# B&R Automation Studio project A2019059_Linka_Power_CP (part 31)

#### Types.typ - Local data types
```iecst
TYPE
	SkrutkovaciSetStruc : 	STRUCT
		VretenoStatus : WSTRING[80];
		VretenoFaza : USINT;
		Zasobnik : ZasobnikStruc;
		Vreteno : VretenoStruc;
		SkrutkaOdobrata : BOOL;
		SkrutkaPripravena : BOOL;
		Manual : BOOL;
		PodajSrobu : BOOL;
		CistenieVykonane : BOOL;
		VykonajCistenie : BOOL;
		Automat : BOOL;
	END_STRUCT;
	INzasobnik : 	STRUCT
		AccumulationSwitch : BOOL; (*Snimac zaplnenia S25*)
		ScrewMeasurement : BOOL; (*Kontrola matice S21*)
		FeederLevelControl : BOOL; (*Hladina v zasobniku S20*)
	END_STRUCT;
	OUTzasobnik : 	STRUCT
		StartA20 : BOOL; (*Zapnutie vibrovania A20*)
		Escapement : BOOL; (*Pustanie matky do hadice Y22*)
		FeedAir : BOOL; (*Strielanie do hadice Y21*)
		SortingAir : BOOL; (*Triedenie kusov Y30*)
		BlowOff : BOOL; (*Zhadzovanie kusov Y25*)
	END_STRUCT;
	INvreteno : 	STRUCT
		ReturnStroke : BOOL; (*Vreteno zasunute S01*)
		DeptControl : BOOL; (*Vreteno vysunute S02*)
		BrakeClosed : BOOL; (*Brzda zatvorena S13*)
		BrakeOpen : BOOL; (*Brzda otvorena S12*)
		ScrewMeasurementBrake : BOOL; (*Kontrola matice pred brzdou S15*)
		ScrewMeasurement : BOOL; (*Kontrola matice v hadici S06*)
	END_STRUCT;
	OUTvreteno : 	STRUCT
		WasteExtraction : BOOL; (*Odstranovanie spiny Y13*)
		Spindle : BOOL; (*Vysunutie vretena Y02*)
		BlastAirBrake : BOOL; (*Strielanie za brzdou Y14*)
		BrakeSpindle : BOOL; (*Brzda vretena Y12*)
		Vacuum : BOOL; (*Pridrzanie skrutky Y15*)
		CounterBlast : BOOL; (*Uvolnenie skrutky Y16*)
	END_STRUCT;
	VretenoStruc : 	STRUCT
		OUT : OUTvreteno;
		IN : INvreteno;
	END_STRUCT;
	ZasobnikStruc : 	STRUCT
		OUT : OUTzasobnik;
		IN : INzasobnik;
	END_STRUCT;
END_TYPE
```

#### Variables.var - Local variables
```iecst
VAR
	Stav_PodavacVycisteny : BOOL;
	Stav_SkrutkaM5_Pripravena : BOOL;
	SkrutkovaciSet : SkrutkovaciSetStruc;
	TprazdnyZasobnik : TON;
	TakumulaciaPlna : TON;
	TvytvorenieVakua : TON;
	TodvetranieVakua : TON;
	TprefukPredBrzdou : TON;
	TvysuvanieSpindle : TON;
	TprefukZaBrzdou : TON;
	PocetPokusovOpripravuSkrutky : USINT;
	ToddelovacZakladnaPoloha : TON;
	TpripravaSkrutky : TON;
	TodsatieNecistot : TON;
	Tvibrovanie : TON;
	TvyfukovaniePredVibrovanim : TON;
	ZapniHrniec : BOOL;
	TpodaniaSkrutky : TON;
	TpredSkrutkaPripravena : TON;
	TvypnutieOfuku : TON;
	StavSkrutkovackaVysunuta : BOOL;
	TalarmuVysunutiaSkrutkovacky : TON;
END_VAR
```

### Program Logical/Program/Pracovisko_2/P2_SkrutkovaciSet_M6 (IEC)

#### Main.st - Init, cyclic, exit code
```iecst
PROGRAM _INIT
    TprazdnyZasobnik.PT:=T#2000ms;
    TakumulaciaPlna.PT:=T#1000ms;
    TvytvorenieVakua.PT:=T#200ms;
    TodvetranieVakua.PT:=T#1s;
    TprefukPredBrzdou.PT:=T#2000ms;
    TprefukZaBrzdou.PT:=T#2000ms;
    TvysuvanieSpindle.PT:=T#1s;
    TpripravaSkrutky.PT:=T#3000ms;
    ToddelovacZakladnaPoloha.PT:=T#1000ms;
    TodsatieNecistot.PT:=T#1000ms;
    Tvibrovanie.PT:=T#3000ms;
    Stav_PodavacVycisteny:= FALSE;
    Stav_SkrutkaM6_Pripravena:= FALSE;
    TvyfukovaniePredVibrovanim.PT:= T#1000ms;
    TpodaniaSkrutky.PT:= T#1000ms;
    TpredSkrutkaPripravena.PT:= T#500ms;
    TvypnutieOfuku.PT:= T#2000ms;
    TalarmuVysunutiaSkrutkovacky.PT:= T#10s;
END_PROGRAM

PROGRAM _CYCLIC

     (********************Mapovanie IN/OUT********************************)

    SkrutkovaciSet.Manual:= P2_Srobovanie.SkrutkovaciSet_M6.Manual;
    SkrutkovaciSet.Automat:= P2_Srobovanie.SkrutkovaciSet_M6.Automat;
    SkrutkovaciSet.SkrutkaOdobrata:=P2_Srobovanie.SkrutkovaciSet_M6.SkrutkaM6_Odobrata;
    P2_Srobovanie.SkrutkovaciSet_M6.SkrutkaM6_Pripravena:= SkrutkovaciSet.SkrutkaPripravena;
    P2_Srobovanie.SkrutkovaciSet_M6.CistenieUkoncene:= SkrutkovaciSet.CistenieVykonane;
    SkrutkovaciSet.VykonajCistenie:= P2_Srobovanie.SkrutkovaciSet_M6.Cistenie;

    SkrutkovaciSet.Vreteno.IN.BrakeClosed:=P2_Srobovanie.IN.SkrutkM6_Cist_BrzdaZatvoren_MS16;
    SkrutkovaciSet.Vreteno.IN.BrakeOpen:=P2_Srobovanie.IN.SkrutkM6_Cist_BrzdaOtvorena_MS15;
    SkrutkovaciSet.Vreteno.IN.DeptControl:=P2_Srobovanie.IN.SkrutkM6_ZASUNUTY_MS14;
    SkrutkovaciSet.Vreteno.IN.ScrewMeasurement:=P2_Srobovanie.IN.SkrutkM6_SrobaPresla_IS38;
    SkrutkovaciSet.Vreteno.IN.ScrewMeasurementBrake:=P2_Srobovanie.IN.SkrutkM6_Cist_SrobaPresla_IS39;

    IF P2_Srobovanie.SkrutkovaciSet_M6.Reset AND SkrutkovaciSet.VretenoFaza <> 102 AND SkrutkovaciSet.VretenoFaza <> 104 THEN
        SkrutkovaciSet.VretenoFaza:=0;
        P2_Srobovanie.SkrutkovaciSet_M6.Reset:= FALSE;
    END_IF

    SkrutkovaciSet.Zasobnik.IN.AccumulationSwitch:=P2_Srobovanie.IN.ZasobSrobM6_ListaPLNA_OS5;
    SkrutkovaciSet.Zasobnik.IN.FeederLevelControl:=P2_Srobovanie.IN.ZasobSrobM6_PRAZDNY_IS36;
    SkrutkovaciSet.Zasobnik.IN.ScrewMeasurement:=P2_Srobovanie.IN.NastrelSrobM6_SrobaPresla_IS37;

    P2_Srobovanie.OUT.SkrutkM6_Cist_OfukVakua_RUN_YV38:=SkrutkovaciSet.Vreteno.OUT.BlastAirBrake;
    P2_Srobovanie.OUT.SkrutkM6_Cist_OTVOR_YV37:=SkrutkovaciSet.Vreteno.OUT.BrakeSpindle;
    P2_Srobovanie.OUT.SkrutkM6_OfukVakua_RUN_YV35:=SkrutkovaciSet.Vreteno.OUT.CounterBlast;
    IF SkrutkovaciSet.VretenoFaza>1 AND SkrutkovaciSet.VretenoFaza<100 THEN
        P2_Srobovanie.OUT.SkrutkM6_VYSUN_YV34:=SkrutkovaciSet.Vreteno.OUT.Spindle;
    END_IF
    P2_Srobovanie.OUT.SkrutkM6_Cist_Vakum_RUN_YV39:=SkrutkovaciSet.Vreteno.OUT.WasteExtraction;
    IF SkrutkovaciSet.VykonajCistenie THEN
        P2_Srobovanie.OUT.SkrutkM6_PrisavSkrutky_RUN_YV36:=SkrutkovaciSet.Vreteno.OUT.Vacuum;
    END_IF
    P2_Srobovanie.OUT.ZasobSrobM6_Ofuk_RUN_YV30:=SkrutkovaciSet.Zasobnik.OUT.BlowOff;
    P2_Srobovanie.OUT.NastrelSrobM6_PosunSrobu_YV32:=SkrutkovaciSet.Zasobnik.OUT.Escapement;
    P2_Srobovanie.OUT.NastrelSrobM6_NastrelSrobu_YV33:=SkrutkovaciSet.Zasobnik.OUT.FeedAir;
    P2_Srobovanie.OUT.ZasobSrobM6_OfukTried_RUN_YV31:=SkrutkovaciSet.Zasobnik.OUT.SortingAir;
    P2_Srobovanie.OUT.ZasobSrobM6_Vibrovanie_RUN_FM2:= SkrutkovaciSet.Zasobnik.OUT.StartA20;

    (********************Časáky********************************)
    TprazdnyZasobnik();
    TakumulaciaPlna();
    TvytvorenieVakua();
    TodvetranieVakua();
    TprefukPredBrzdou();
    TprefukZaBrzdou();
    TvysuvanieSpindle();
    TpripravaSkrutky();
    ToddelovacZakladnaPoloha();
    TodsatieNecistot();
    Tvibrovanie();
    TvyfukovaniePredVibrovanim();
    TpodaniaSkrutky();
    TpredSkrutkaPripravena();
    TvypnutieOfuku();
    TalarmuVysunutiaSkrutkovacky();
    (********************Zásobnik********************************)

    //kontrola akumulacie
    IF SkrutkovaciSet.Zasobnik.IN.AccumulationSwitch=1 THEN
        TakumulaciaPlna.IN:=1;
    ELSE
        TakumulaciaPlna.IN:=0;
    END_IF

    //kontrola naplnenia zasobnika
    IF SkrutkovaciSet.Zasobnik.IN.FeederLevelControl=1 THEN
        TprazdnyZasobnik.IN:=1;
    ELSE
        TprazdnyZasobnik.IN:=0;
    END_IF

    //Ovládanie vzduchov zásobníka//
    IF ZapniHrniec THEN
        IF TakumulaciaPlna.Q=1 THEN
            SkrutkovaciSet.Zasobnik.OUT.BlowOff:=1;
        ELSE
            SkrutkovaciSet.Zasobnik.OUT.BlowOff:=0;
        END_IF
        SkrutkovaciSet.Zasobnik.OUT.SortingAir:= 1;
    ELSE
        SkrutkovaciSet.Zasobnik.OUT.BlowOff:=0;
    END_IF

    IF NOT SkrutkovaciSet.Zasobnik.OUT.StartA20 AND NOT ZapniHrniec THEN
        TvypnutieOfuku.IN:= 1;
    ELSE
        TvypnutieOfuku.IN:= 0;
    END_IF

    IF EDGEPOS(TvypnutieOfuku.Q) THEN
        SkrutkovaciSet.Zasobnik.OUT.SortingAir:= 0;
    END_IF

    //ovladanie vibracneho podavaca
    IF ZapniHrniec THEN
        TvyfukovaniePredVibrovanim.IN:= 1;
    ELSE
        TvyfukovaniePredVibrovanim.IN:= 0;
    END_IF

    IF ZapniHrniec AND TvyfukovaniePredVibrovanim.Q THEN
        SkrutkovaciSet.Zasobnik.OUT.StartA20:=1;
        Tvibrovanie.IN:=1;
    ELSE
        SkrutkovaciSet.Zasobnik.OUT.StartA20:=0;
        Tvibrovanie.IN:=0;
    END_IF

    IF Tvibrovanie.Q=1 THEN
        IF TakumulaciaPlna.Q=1 AND NOT P2_Srobovanie.RR_ZapniHrniec_M6 THEN
            ZapniHrniec:= 0;
        END_IF
    END_IF

    //Zapnutie hrnca v ručnom režime//
    IF EDGEPOS(P2_Srobovanie.RR_ZapniHrniec_M6) THEN
        ZapniHrniec:= TRUE;
    END_IF
    IF EDGENEG(P2_Srobovanie.RR_ZapniHrniec_M6) THEN
        ZapniHrniec:= FALSE;
    END_IF

    //Zrušenie signálu skrutka pripravená//
    IF SkrutkovaciSet.SkrutkaPripravena=1 THEN
        IF SkrutkovaciSet.SkrutkaOdobrata=1 THEN
            SkrutkovaciSet.SkrutkaPripravena:=0;
        END_IF
    END_IF

    (********************Vreteno********************************)
    CASE SkrutkovaciSet.VretenoFaza OF
        0: SkrutkovaciSet.VretenoStatus:="Vypnute";
            SkrutkovaciSet.Vreteno.OUT.BlastAirBrake:=0;
            SkrutkovaciSet.Vreteno.OUT.BrakeSpindle:=0;
            SkrutkovaciSet.Vreteno.OUT.CounterBlast:=0;
            SkrutkovaciSet.Vreteno.OUT.Spindle:=0;
            SkrutkovaciSet.Vreteno.OUT.Vacuum:=0;
            SkrutkovaciSet.Vreteno.OUT.WasteExtraction:=0;

            SkrutkovaciSet.Zasobnik.OUT.Escapement:=0;
            SkrutkovaciSet.Zasobnik.OUT.FeedAir:=0;

            SkrutkovaciSet.Zasobnik.OUT.StartA20:=0;

            SkrutkovaciSet.CistenieVykonane:=0;
            SkrutkovaciSet.SkrutkaPripravena:=0;

            TprazdnyZasobnik.IN:=0;
            TakumulaciaPlna.IN:=0;
            TvytvorenieVakua.IN:=0;
            TodvetranieVakua.IN:=0;
            TprefukPredBrzdou.IN:=0;
            TprefukZaBrzdou.IN:=0;
            TvysuvanieSpindle.IN:=0;
            TpripravaSkrutky.IN:=0;
            ToddelovacZakladnaPoloha.IN:=0;
            TodsatieNecistot.IN:=0;
            TpodaniaSkrutky.IN:= 0;
            TpredSkrutkaPripravena.IN:= 0;
            ZapniHrniec:= 0;
            PocetPokusovOpripravuSkrutky:=0;
            StavSkrutkovackaVysunuta:= 0;
            TalarmuVysunutiaSkrutkovacky.IN:= 0;
            SkrutkovaciSet.VretenoFaza:=1;

        1: SkrutkovaciSet.VretenoStatus:="Inicializacia: cakam na povel";
            IF SkrutkovaciSet.Automat=1 THEN
                SkrutkovaciSet.CistenieVykonane:=0;
                SkrutkovaciSet.SkrutkaPripravena:=0;
                SkrutkovaciSet.VretenoFaza:=2;
            ELSIF SkrutkovaciSet.Manual=1 THEN
                SkrutkovaciSet.VretenoFaza:=250;
            END_IF

        2: SkrutkovaciSet.VretenoStatus:="Inicializacia: cakam na povel precisti hadice";

            IF SkrutkovaciSet.VykonajCistenie=1 THEN
                SkrutkovaciSet.Vreteno.OUT.Vacuum:=1;
                SkrutkovaciSet.VretenoFaza:=3;
            END_IF

        3: SkrutkovaciSet.VretenoStatus:="Inicializacia: Cakam na snimac: vreteno vysunute";
            SkrutkovaciSet.Vreteno.OUT.Spindle:=1;
            TalarmuVysunutiaSkrutkovacky.IN:= 1;

            IF P2_Srobovanie.IN.SkrutkM6_VysunutieHrotu_IOS3 > 1 THEN
                StavSkrutkovackaVysunuta:= TRUE;
                TvysuvanieSpindle.IN:=1;
            END_IF

            IF TvysuvanieSpindle.Q=1 AND StavSkrutkovackaVysunuta THEN
                TodvetranieVakua.IN:= 1;
                SkrutkovaciSet.Vreteno.OUT.CounterBlast:=1;
                SkrutkovaciSet.Vreteno.OUT.Vacuum:=0;
            END_IF

            IF TvysuvanieSpindle.Q AND StavSkrutkovackaVysunuta AND TodvetranieVakua.Q THEN
                StavSkrutkovackaVysunuta:= FALSE;
                TalarmuVysunutiaSkrutkovacky.IN:= 0;
                TvysuvanieSpindle.IN:=0;
                TodvetranieVakua.IN:= 0;
                SkrutkovaciSet.VretenoFaza:=4;
            ELSIF TalarmuVysunutiaSkrutkovacky.Q THEN
                P2_Alarmy[270]:= TRUE;
                P2_PoruchaST3:= TRUE;
            END_IF

        4: SkrutkovaciSet.VretenoStatus:="Inicializacia: Cakam na snimac: vreteno zasunute";
            SkrutkovaciSet.Vreteno.OUT.Spindle:=0;
            IF SkrutkovaciSet.Vreteno.IN.DeptControl=1 THEN
                SkrutkovaciSet.Vreteno.OUT.CounterBlast:=0;
                SkrutkovaciSet.VretenoFaza:=5;
            END_IF

        5: SkrutkovaciSet.VretenoStatus:="Inicializacia: Cakam na prefuknutie hadice za brzdou";
            TprefukZaBrzdou.IN:=1;
            SkrutkovaciSet.Vreteno.OUT.BlastAirBrake:=1;
            IF TprefukZaBrzdou.Q=1 THEN
                TprefukZaBrzdou.IN:=0;
                SkrutkovaciSet.Vreteno.OUT.BlastAirBrake:=0;
                SkrutkovaciSet.VretenoFaza:=6;
            END_IF

        6: SkrutkovaciSet.VretenoStatus:="Inicializacia: vypinam prefuk";
            TprefukZaBrzdou.IN:=0;
            SkrutkovaciSet.Vreteno.OUT.BlastAirBrake:=0;
            SkrutkovaciSet.Vreteno.OUT.Vacuum:=1;
            SkrutkovaciSet.VretenoFaza:=7;

        7: SkrutkovaciSet.VretenoStatus:="Inicializacia: Cakam na snimac: vreteno vysunute";
            SkrutkovaciSet.Vreteno.OUT.Spindle:=1;
            TalarmuVysunutiaSkrutkovacky.IN:= 1;

            IF P2_Srobovanie.IN.SkrutkM6_VysunutieHrotu_IOS3 > 1 THEN
                StavSkrutkovackaVysunuta:= TRUE;
                TvysuvanieSpindle.IN:=1;
            END_IF

            IF TvysuvanieSpindle.Q=1 AND StavSkrutkovackaVysunuta THEN
                TodvetranieVakua.IN:= 1;
                SkrutkovaciSet.Vreteno.OUT.CounterBlast:=1;
                SkrutkovaciSet.Vreteno.OUT.Vacuum:=0;
            END_IF

            IF TvysuvanieSpindle.Q AND StavSkrutkovackaVysunuta AND TodvetranieVakua.Q THEN
                StavSkrutkovackaVysunuta:= FALSE;
                TalarmuVysunutiaSkrutkovacky.IN:= 0;
                TvysuvanieSpindle.IN:=0;
                TodvetranieVakua.IN:= 0;
                SkrutkovaciSet.VretenoFaza:=8;
            ELSIF TalarmuVysunutiaSkrutkovacky.Q THEN
                P2_Alarmy[270]:= TRUE;
                P2_PoruchaST3:= TRUE;
            END_IF

        8: SkrutkovaciSet.VretenoStatus:="Inicializacia: Cakam na snimac: vreteno zasunute";
            SkrutkovaciSet.Vreteno.OUT.Spindle:=0;
            IF SkrutkovaciSet.Vreteno.IN.DeptControl=1 THEN
                SkrutkovaciSet.Vreteno.OUT.CounterBlast:=0;
                SkrutkovaciSet.VretenoFaza:=9;
            END_IF

        9: SkrutkovaciSet.VretenoStatus:="Inicializacia: Cakam na prefuknutie hadice pred brzdou";
            TprefukPredBrzdou.IN:=1;
            SkrutkovaciSet.Zasobnik.OUT.FeedAir:=1;
            IF TprefukPredBrzdou.Q=1 THEN
                TprefukPredBrzdou.IN:=0;
                SkrutkovaciSet.Zasobnik.OUT.FeedAir:=0;
                SkrutkovaciSet.VretenoFaza:=10;
            END_IF

        10: SkrutkovaciSet.VretenoStatus:="Inicializacia: Cakam na snimac: brzda uvolnena";
            SkrutkovaciSet.Vreteno.OUT.BrakeSpindle:=1;
            IF SkrutkovaciSet.Vreteno.IN.BrakeOpen=1 THEN
                SkrutkovaciSet.Vreteno.OUT.BlastAirBrake:=1;
                SkrutkovaciSet.VretenoFaza:=11;
            END_IF

        11: SkrutkovaciSet.VretenoStatus:="Inicializacia: Cakam na prefuknutie hadice za brzdou";
            TprefukZaBrzdou.IN:=1;
            SkrutkovaciSet.Vreteno.OUT.BlastAirBrake:=1;
            IF TprefukZaBrzdou.Q=1 THEN
                TprefukZaBrzdou.IN:=0;
                SkrutkovaciSet.Vreteno.OUT.BlastAirBrake:=0;
                SkrutkovaciSet.VretenoFaza:=12;
            END_IF

        12: SkrutkovaciSet.VretenoStatus:="Inicializacia: vypinam prefuk";
            TprefukZaBrzdou.IN:=0;
            SkrutkovaciSet.Vreteno.OUT.BlastAirBrake:=0;
            SkrutkovaciSet.Vreteno.OUT.Vacuum:=1;
            SkrutkovaciSet.VretenoFaza:=13;

        13: SkrutkovaciSet.VretenoStatus:="Inicializacia: Cakam na snimac: vreteno vysunute";
            SkrutkovaciSet.Vreteno.OUT.Spindle:=1;
            TalarmuVysunutiaSkrutkovacky.IN:= 1;

            IF P2_Srobovanie.IN.SkrutkM6_VysunutieHrotu_IOS3 > 1 THEN
                StavSkrutkovackaVysunuta:= TRUE;
                TvysuvanieSpindle.IN:=1;
            END_IF

            IF TvysuvanieSpindle.Q=1 AND StavSkrutkovackaVysunuta THEN
                TodvetranieVakua.IN:= 1;
                SkrutkovaciSet.Vreteno.OUT.CounterBlast:=1;
                SkrutkovaciSet.Vreteno.OUT.Vacuum:=0;
            END_IF

            IF TvysuvanieSpindle.Q AND StavSkrutkovackaVysunuta AND TodvetranieVakua.Q THEN
                StavSkrutkovackaVysunuta:= FALSE;
                TalarmuVysunutiaSkrutkovacky.IN:= 0;
                TvysuvanieSpindle.IN:=0;
                TodvetranieVakua.IN:= 0;
                SkrutkovaciSet.VretenoFaza:=14;
            ELSIF TalarmuVysunutiaSkrutkovacky.Q THEN
                P2_Alarmy[270]:= TRUE;
                P2_PoruchaST3:= TRUE;
            END_IF

        14: SkrutkovaciSet.VretenoStatus:="Inicializacia: Cakam na snimac: vreteno zasunute";
            SkrutkovaciSet.Vreteno.OUT.Spindle:=0;
            IF SkrutkovaciSet.Vreteno.IN.DeptControl=1 THEN
                SkrutkovaciSet.Vreteno.OUT.CounterBlast:=0;
                SkrutkovaciSet.VretenoFaza:=15;
            END_IF

        15: SkrutkovaciSet.VretenoStatus:="Inicializacia: Cakam na snimac: brzda zasunuta";
            SkrutkovaciSet.Vreteno.OUT.BrakeSpindle:=0;
            IF SkrutkovaciSet.Vreteno.IN.BrakeClosed=1 THEN
                SkrutkovaciSet.CistenieVykonane:=1;
                SkrutkovaciSet.VretenoFaza:=16;
            END_IF

        16: SkrutkovaciSet.VretenoStatus:="Inicializacia: Cakam na zrusenie signalu: vykonaj cistenie";
            IF SkrutkovaciSet.VykonajCistenie=0 THEN
                SkrutkovaciSet.CistenieVykonane:=0;
                SkrutkovaciSet.SkrutkaPripravena:=0;
                SkrutkovaciSet.VretenoFaza:=100;
            END_IF

        100: SkrutkovaciSet.VretenoStatus:="Cakam kym zasobnik pripravy skrutku";
            ZapniHrniec:= 1;
            IF TakumulaciaPlna.Q=1 AND SkrutkovaciSet.Zasobnik.OUT.StartA20 THEN
                TpodaniaSkrutky.IN:= 1;
            END_IF

            IF TpodaniaSkrutky.Q THEN
                TpodaniaSkrutky.IN:= 0;
                SkrutkovaciSet.VretenoFaza:=102;
            END_IF

        102: SkrutkovaciSet.VretenoStatus:="Cakam na snimac: skrutka presla hadicou";
            SkrutkovaciSet.Zasobnik.OUT.Escapement:=1;
            TpripravaSkrutky.IN:=1;
            IF SkrutkovaciSet.Zasobnik.IN.ScrewMeasurement=1 THEN
                SkrutkovaciSet.Zasobnik.OUT.FeedAir:=1;
                TpripravaSkrutky.IN:=0;
                SkrutkovaciSet.VretenoFaza:=104;
            ELSIF TpripravaSkrutky.Q=1 THEN
                TpripravaSkrutky.IN:=0;
                SkrutkovaciSet.Zasobnik.OUT.Escapement:=0;
                SkrutkovaciSet.VretenoFaza:=100;
            END_IF

        104: SkrutkovaciSet.VretenoStatus:="Cakam na snimac: skrutka presla hadicou pred brzdou";
            IF SkrutkovaciSet.Vreteno.IN.ScrewMeasurementBrake=1 THEN
                SkrutkovaciSet.Zasobnik.OUT.Escapement:=0;
                SkrutkovaciSet.Zasobnik.OUT.FeedAir:=0;
                PocetPokusovOpripravuSkrutky:=0;
                SkrutkovaciSet.VretenoFaza:=106;
            END_IF

        106: SkrutkovaciSet.VretenoStatus:="Cakam na odsatie necistot";
            SkrutkovaciSet.Vreteno.OUT.WasteExtraction:=1;
            TodsatieNecistot.IN:=1;

            IF TodsatieNecistot.Q=1 THEN
                TodsatieNecistot.IN:=0;
                SkrutkovaciSet.Vreteno.OUT.WasteExtraction:=0;
                SkrutkovaciSet.VretenoFaza:=107;
            END_IF

        107: SkrutkovaciSet.VretenoStatus:="Cakam kym skrutkovacka odoberie skrutku";
            IF SkrutkovaciSet.SkrutkaPripravena=0 AND SkrutkovaciSet.SkrutkaOdobrata=0 THEN
                SkrutkovaciSet.VretenoFaza:=108;
            END_IF

        108: SkrutkovaciSet.VretenoStatus:="Cakam na snimac: brzda uvolnena";
            SkrutkovaciSet.Vreteno.OUT.BrakeSpindle:=1;
            IF SkrutkovaciSet.Vreteno.IN.BrakeOpen=1 THEN
                SkrutkovaciSet.Vreteno.OUT.BlastAirBrake:=1;
                SkrutkovaciSet.VretenoFaza:=110;
            END_IF

        110: SkrutkovaciSet.VretenoStatus:="Cakam na snimac: skrutka presla hadicou pred vretenom";
            IF SkrutkovaciSet.Vreteno.IN.ScrewMeasurement=1 THEN
                SkrutkovaciSet.Vreteno.OUT.BlastAirBrake:=0;
                SkrutkovaciSet.Vreteno.OUT.BrakeSpindle:=0;
                SkrutkovaciSet.VretenoFaza:=112;
            END_IF

        112: SkrutkovaciSet.VretenoStatus:="Cakam na snimac: brzda zabrzdena";
            SkrutkovaciSet.Vreteno.OUT.BrakeSpindle:=0;
            IF SkrutkovaciSet.Vreteno.IN.BrakeClosed=1 AND SkrutkovaciSet.SkrutkaOdobrata=0 THEN
                TpredSkrutkaPripravena.IN:= 1;
                IF TpredSkrutkaPripravena.Q THEN
                    TpredSkrutkaPripravena.IN:= 0;
                    SkrutkovaciSet.SkrutkaPripravena:=1;
                    SkrutkovaciSet.VretenoFaza:=100;
                END_IF
            END_IF

            //*************** opakovany pokus o oddelenie skrutky *********************************

        170: SkrutkovaciSet.VretenoStatus:="Cakam na presunutie oddelovaca do zakladnej polohy";
            SkrutkovaciSet.Zasobnik.OUT.Escapement:=0;
            ToddelovacZakladnaPoloha.IN:=1;
            IF ToddelovacZakladnaPoloha.Q=1 THEN
                ToddelovacZakladnaPoloha.IN:=0;
                PocetPokusovOpripravuSkrutky:=PocetPokusovOpripravuSkrutky+1;
                IF PocetPokusovOpripravuSkrutky>3 THEN
                    PocetPokusovOpripravuSkrutky:=0;
                    SkrutkovaciSet.VretenoFaza:=171;
                ELSE
                    SkrutkovaciSet.VretenoFaza:=100;
                END_IF
            END_IF

        171: SkrutkovaciSet.VretenoStatus:="Zaseknuta skrutka v oddelovaci!!!";
    END_CASE

END_PROGRAM

PROGRAM _EXIT
	(* Insert code here *)

END_PROGRAM
```

#### Types.typ - Local data types
```iecst
TYPE
	SkrutkovaciSetStruc : 	STRUCT
		VretenoStatus : WSTRING[80];
		VretenoFaza : USINT;
		Zasobnik : ZasobnikStruc;
		Vreteno : VretenoStruc;
		SkrutkaOdobrata : BOOL;
		SkrutkaPripravena : BOOL;
		Manual : BOOL;
		PodajSrobu : BOOL;
		CistenieVykonane : BOOL;
		VykonajCistenie : BOOL;
		Automat : BOOL;
	END_STRUCT;
	INzasobnik : 	STRUCT
		AccumulationSwitch : BOOL; (*Snimac zaplnenia S25*)
		ScrewMeasurement : BOOL; (*Kontrola matice S21*)
		FeederLevelControl : BOOL; (*Hladina v zasobniku S20*)
	END_STRUCT;
	OUTzasobnik : 	STRUCT
		StartA20 : BOOL; (*Zapnutie vibrovania A20*)
		Escapement : BOOL; (*Pustanie matky do hadice Y22*)
		FeedAir : BOOL; (*Strielanie do hadice Y21*)
		SortingAir : BOOL; (*Triedenie kusov Y30*)
		BlowOff : BOOL; (*Zhadzovanie kusov Y25*)
	END_STRUCT;
	INvreteno : 	STRUCT
		ReturnStroke : BOOL; (*Vreteno zasunute S01*)
		DeptControl : BOOL; (*Vreteno vysunute S02*)
		BrakeClosed : BOOL; (*Brzda zatvorena S13*)
		BrakeOpen : BOOL; (*Brzda otvorena S12*)
		ScrewMeasurementBrake : BOOL; (*Kontrola matice pred brzdou S15*)
		ScrewMeasurement : BOOL; (*Kontrola matice v hadici S06*)
	END_STRUCT;
	OUTvreteno : 	STRUCT
		WasteExtraction : BOOL; (*Odstranovanie spiny Y13*)
		Spindle : BOOL; (*Vysunutie vretena Y02*)
		BlastAirBrake : BOOL; (*Strielanie za brzdou Y14*)
		BrakeSpindle : BOOL; (*Brzda vretena Y12*)
		Vacuum : BOOL; (*Pridrzanie skrutky Y15*)
		CounterBlast : BOOL; (*Uvolnenie skrutky Y16*)
	END_STRUCT;
	VretenoStruc : 	STRUCT
		OUT : OUTvreteno;
		IN : INvreteno;
	END_STRUCT;
	ZasobnikStruc : 	STRUCT
		OUT : OUTzasobnik;
		IN : INzasobnik;
	END_STRUCT;
END_TYPE
```

#### Variables.var - Local variables
```iecst
VAR
	Stav_PodavacVycisteny : BOOL;
	Stav_SkrutkaM6_Pripravena : BOOL;
	SkrutkovaciSet : SkrutkovaciSetStruc;
	TprazdnyZasobnik : TON;
	TakumulaciaPlna : TON;
	TvytvorenieVakua : TON;
	TodvetranieVakua : TON;
	TprefukPredBrzdou : TON;
	TvysuvanieSpindle : TON;
	TprefukZaBrzdou : TON;
	PocetPokusovOpripravuSkrutky : USINT;
	ToddelovacZakladnaPoloha : TON;
	TpripravaSkrutky : TON;
	TodsatieNecistot : TON;
	Tvibrovanie : TON;
	TvyfukovaniePredVibrovanim : TON;
	ZapniHrniec : BOOL;
	TpodaniaSkrutky : TON;
	TpredSkrutkaPripravena : TON;
	TvypnutieOfuku : TON;
	StavSkrutkovackaVysunuta : BOOL;
	TalarmuVysunutiaSkrutkovacky : TON;
END_VAR
```

### Program Logical/Program/Pracovisko_2/P2_Robot (IEC)

#### Main.st - Init, cyclic, exit code
```iecst
PROGRAM _INIT
	Triger_0:= FALSE;

END_PROGRAM

PROGRAM _CYCLIC

	//Volanie funkcie SequenceControl//
	SequenceControl(SC:= SC_P2_Robot);

	//Volanie podprogramov//
	IOLinkKomunikacia;
	ProfinetKomunikaciaRobot;

	//Reset sekcie //
	IF NOT Safety.STAV.ZonaCS_AKTIVNA THEN
		SC_P2_Robot.Step:= 0;
	ELSIF P2_PoruchaST3 AND NOT P2_StoperSrobovania.Automat AND NOT P2_StoperZvarania.Automat THEN
		SC_P2_Robot.Step:= 0;
	ELSIF P2_PoruchaST4 AND NOT P2_StoperSrobovania.Automat AND NOT P2_StoperZvarania.Automat THEN
		SC_P2_Robot.Step:= 0;
	ELSIF P2_Robot.Reset THEN
		SC_P2_Robot.Step:= 0;
		P2_Robot.Reset:= FALSE;
	END_IF

    IF NOT Safety.STAV.P2_ZonaBunky_AKTIVNA AND NOT Triger_0 THEN
        Triger_0:= TRUE;
        SC_P2_Robot.Step:= 0;
    END_IF

    IF Safety.STAV.P2_ZonaBunky_AKTIVNA THEN
        Triger_0:= FALSE;
    END_IF

	CASE SC_P2_Robot.Step OF

		0:
			SC_P2_Robot.StepName:='0 - Nulovanie';
			P2_Robot.Automat:= FALSE;
			P2_Robot.KoniecCyklu:= FALSE;
			P2_Robot.Manual:= FALSE;
			P2_Robot.Reset:= FALSE;
			P2_Robot.STAV.PoINIT:= FALSE;
			P2_Robot.KOM_OUT.Odparkovanie:= FALSE;
			P2_Robot.KOM_OUT.PP_na_Main:= FALSE;
			P2_Robot.KOM_OUT.Reset_CS:= FALSE;
			P2_Robot.KOM_OUT.StartProgramu:= FALSE;
			P2_Robot.KOM_OUT.StartProgramuMain:= FALSE;
			P2_Robot.KOM_OUT.VypniMotory:= FALSE;
			P2_Robot.KOM_OUT.ZapniMotory:= FALSE;
			IF P2_Robot.KOM_IN.Stav_RezimAUTOMAT AND P2_Robot.KOM_IN.Stav_ProgramRUN THEN
				P2_Robot.KOM_OUT.StopProgramu:= TRUE;
			ELSE
				P2_Robot.KOM_OUT.StopProgramu:= FALSE;
			END_IF
			IF Safety.STAV.ZonaCS_AKTIVNA AND Safety.STAV.P2_ZonaBunky_AKTIVNA AND NOT P2_Pracovisko.STAV.PORUCHA AND P2_Pracovisko.IN.PrivodVzduchu_SnimacTlaku_S3 AND NOT P2_Robot.KOM_IN.Stav_ProgramRUN THEN
				P2_Robot.KOM_OUT.StopProgramu:= FALSE;
				SC_P2_Robot.ResetStep:= TRUE;
				SC_P2_Robot.Step:= 1;
			END_IF

		1:
			SC_P2_Robot.StepName:='1 - Cakam na spustenie vyroby';
			P2_Robot.KoniecCyklu:= FALSE;
            IF P2_Robot.Automat THEN
				SC_P2_Robot.Step:= 2;
			ELSIF P2_Robot.Manual THEN
				SC_P2_Robot.Step:= 700;
			END_IF

		//********************************************************Inicializácia****************************************************************************//

		2:
			SC_P2_Robot.StepName:='2 - Inicializacia - cakam na spustenie inicializacie';
			SC_P2_Robot.IdleTime.PT:= T#500ms;
			SC_P2_Robot.AlarmTime.PT:= T#5s;

			SC_P2_Robot.IdleTime.IN:= TRUE;

			IF SC_P2_Robot.IdleTime.Q THEN
				SC_P2_Robot.ResetStep:= TRUE;
				SC_P2_Robot.Step:= 3;
			END_IF

		3:
			SC_P2_Robot.StepName:='2 - Inicializacia - kontrolujem central stop robota';
			SC_P2_Robot.IdleTime.PT:= T#500ms;
			SC_P2_Robot.AlarmTime.PT:= T#5s;

			IF P2_Robot.KOM_IN.Stav_RobotCS THEN
				P2_Robot.KOM_OUT.Reset_CS:= TRUE;
			END_IF

			IF NOT P2_Robot.KOM_IN.Stav_RobotCS THEN
				P2_Robot.KOM_OUT.Reset_CS:= FALSE;
				SC_P2_Robot.ResetStep:= TRUE;
				SC_P2_Robot.Step:= 4;
			END_IF

		4:
			SC_P2_Robot.StepName:='4 - Inicializacia - zapinam motory robota';
			SC_P2_Robot.IdleTime.PT:= T#5s;
            SC_P2_Robot.AlarmTime.PT:= T#5s;
            SC_P2_Robot.IdleTime.IN:= TRUE;

			IF NOT P2_Robot.KOM_IN.Stav_MotoryON THEN
				P2_Robot.KOM_OUT.ZapniMotory:= TRUE;
			END_IF

			IF P2_Robot.KOM_IN.Stav_MotoryON OR SC_P2_Robot.IdleTime.Q THEN
				P2_Robot.KOM_OUT.ZapniMotory:= FALSE;
				SC_P2_Robot.ResetStep:= TRUE;
				SC_P2_Robot.Step:= 6;
			END_IF

		6:
			SC_P2_Robot.StepName:='6 - Inicializacia - spustam program robota od zaciatku';
			SC_P2_Robot.IdleTime.PT:= T#500ms;
			SC_P2_Robot.AlarmTime.PT:= T#5s;

			IF NOT SC_P2_Robot.Switch1 THEN
				P2_Robot.KOM_OUT.StartProgramuMain:= TRUE;
				SC_P2_Robot.Switch1:= TRUE;
			END_IF

			IF P2_Robot.KOM_IN.Stav_ProgramRUN (*AND P2_Robot.KOM_IN.Stav_VystupyZresetovane*) THEN
				P2_Robot.KOM_OUT.StartProgramuMain:= FALSE;
				P2_Robot.STAV.PoINIT:= TRUE;
				SC_P2_Robot.ResetStep:= TRUE;
				SC_P2_Robot.Step:= 100;
			END_IF

			//********************************************************Automatický režim****************************************************************************//

		100:
			SC_P2_Robot.StepName:='100 - Automaticky Rezim - cakam na ukoncenie programu robota';
			SC_P2_Robot.IdleTime.PT:= T#200ms;
			SC_P2_Robot.AlarmTime.PT:= T#5s;

			IF P2_Robot.KoniecCyklu AND NOT P2_StoperSrobovania.Automat AND NOT P2_StoperZvarania.Automat AND P2_Robot.KOM_IN.Stav_RobotOdparkovany THEN
                SC_P2_Robot.ResetStep:= TRUE;
                SC_P2_Robot.Step:= 0;
            END_IF

            //*******************************************************Manuálny režim*******************************************************************************//

        700:
			SC_P2_Robot.StepName:='700 - Manualny Rezim';
			SC_P2_Robot.IdleTime.PT:= T#8s;
			SC_P2_Robot.AlarmTime.PT:= T#5s;

	END_CASE

END_PROGRAM

PROGRAM _EXIT
	(* Insert code here *)

END_PROGRAM
```

#### Variables.var - Local variables
```iecst
VAR
	Triger_0 : BOOL;
	CasOtvoreniaGripraMV : TON;
END_VAR
```

#### IOLinkKomunikacia.st
```iecst
ACTION IOLinkKomunikacia:

	//Modul ovládania gripra//
	P2_Robot.IN.GriperMvCase_Otvoreny_IS4:=	P2_Robot.PAR.Modul_IOLink_Inputs.0;
	P2_Robot.IN.GriperMvCase_DrziPowerCP_IS5:=	P2_Robot.PAR.Modul_IOLink_Inputs.1;
	P2_Robot.IN.GriperMvCase_DrziMVcase_IS6:= P2_Robot.PAR.Modul_IOLink_Inputs.2;
	P2_Robot.PAR.Modul_IOLink_Inputs.3;
	P2_Robot.PAR.Modul_IOLink_Inputs.4;
	P2_Robot.PAR.Modul_IOLink_Inputs.5;
	P2_Robot.IN.KodGripra_Bit0:= P2_Robot.PAR.Modul_IOLink_Inputs.6;
	P2_Robot.IN.KodGripra_Bit1:= P2_Robot.PAR.Modul_IOLink_Inputs.7;

	//Kodovanie griprov//
	IF P2_Robot.IN.KodGripra_Bit0 AND P2_Robot.IN.KodGripra_Bit1 THEN
		P2_Robot.KOM_OUT.TypGripra_MV:= FALSE;
		P2_Robot.KOM_OUT.TypGripra_45F:= FALSE;
		P2_Robot.KOM_OUT.TypGripra_5H:= TRUE;
	ELSIF NOT P2_Robot.IN.KodGripra_Bit0 AND P2_Robot.IN.KodGripra_Bit1 THEN
		P2_Robot.KOM_OUT.TypGripra_MV:= FALSE;
		P2_Robot.KOM_OUT.TypGripra_5H:= FALSE;
		P2_Robot.KOM_OUT.TypGripra_45F:= TRUE;
	ELSIF P2_Robot.IN.KodGripra_Bit0 AND NOT P2_Robot.IN.KodGripra_Bit1 THEN
		P2_Robot.KOM_OUT.TypGripra_5H:= FALSE;
		P2_Robot.KOM_OUT.TypGripra_45F:= FALSE;
		P2_Robot.KOM_OUT.TypGripra_MV:= TRUE;
	ELSE
		P2_Robot.KOM_OUT.TypGripra_MV:= FALSE;
		P2_Robot.KOM_OUT.TypGripra_5H:= FALSE;
		P2_Robot.KOM_OUT.TypGripra_45F:= FALSE;
	END_IF

	//Stavy griprov//
	IF P2_Robot.KOM_OUT.TypGripra_45F THEN
		IF P2_Robot.PAR.Griper_4F_5F_5H_IOLink_Inputs <= 30 THEN
			P2_Robot.KOM_OUT.Griper4F_DrziBusbary:= FALSE;
			P2_Robot.KOM_OUT.Griper4F_Zatvoreny:= FALSE;
			P2_Robot.KOM_OUT.Griper4F_Otvoreny:= TRUE;
		ELSIF P2_Robot.PAR.Griper_4F_5F_5H_IOLink_Inputs >= 803 AND P2_Robot.PAR.Griper_4F_5F_5H_IOLink_Inputs <= 900 THEN
			P2_Robot.KOM_OUT.Griper4F_Otvoreny:= FALSE;
			P2_Robot.KOM_OUT.Griper4F_Zatvoreny:= FALSE;
			P2_Robot.KOM_OUT.Griper4F_DrziBusbary:= TRUE;
		ELSIF P2_Robot.PAR.Griper_4F_5F_5H_IOLink_Inputs >= 990 THEN
			P2_Robot.KOM_OUT.Griper4F_Otvoreny:= FALSE;
			P2_Robot.KOM_OUT.Griper4F_DrziBusbary:= FALSE;
			P2_Robot.KOM_OUT.Griper4F_Zatvoreny:= TRUE;
		ELSE
			P2_Robot.KOM_OUT.Griper4F_Otvoreny:= FALSE;
			P2_Robot.KOM_OUT.Griper4F_DrziBusbary:= FALSE;
			P2_Robot.KOM_OUT.Griper4F_Zatvoreny:= FALSE;
		END_IF
	ELSIF P2_Robot.KOM_OUT.TypGripra_MV THEN
		IF P2_Robot.IN.GriperMvCase_Otvoreny_IS4 AND NOT P2_Robot.IN.GriperMvCase_DrziPowerCP_IS5 AND NOT P2_Robot.IN.GriperMvCase_DrziMVcase_IS6 THEN
			P2_Robot.KOM_OUT.GriperMvCase_DrziMVcase:= FALSE;
			P2_Robot.KOM_OUT.GriperMvCase_DrziPowerCP:= FALSE;
			P2_Robot.KOM_OUT.GriperMvCase_Zatvoreny:= FALSE;
			P2_Robot.KOM_OUT.GriperMvCase_Otvoreny:= TRUE;
		ELSIF NOT P2_Robot.IN.GriperMvCase_Otvoreny_IS4 AND P2_Robot.IN.GriperMvCase_DrziPowerCP_IS5 AND P2_Robot.IN.GriperMvCase_DrziMVcase_IS6 THEN
			P2_Robot.KOM_OUT.GriperMvCase_Otvoreny:= FALSE;
			P2_Robot.KOM_OUT.GriperMvCase_DrziPowerCP:= FALSE;
			P2_Robot.KOM_OUT.GriperMvCase_Zatvoreny:= FALSE;
			P2_Robot.KOM_OUT.GriperMvCase_DrziMVcase:= TRUE;
		ELSIF P2_Robot.IN.GriperMvCase_Otvoreny_IS4 AND P2_Robot.IN.GriperMvCase_DrziPowerCP_IS5 AND NOT P2_Robot.IN.GriperMvCase_DrziMVcase_IS6 THEN
			P2_Robot.KOM_OUT.GriperMvCase_Otvoreny:= FALSE;
			P2_Robot.KOM_OUT.GriperMvCase_DrziMVcase:= FALSE;
			P2_Robot.KOM_OUT.GriperMvCase_Zatvoreny:= FALSE;
			P2_Robot.KOM_OUT.GriperMvCase_DrziPowerCP:= TRUE;
		ELSIF NOT P2_Robot.IN.GriperMvCase_Otvoreny_IS4 AND P2_Robot.IN.GriperMvCase_DrziPowerCP_IS5 AND NOT P2_Robot.IN.GriperMvCase_DrziMVcase_IS6 THEN
			P2_Robot.KOM_OUT.GriperMvCase_Otvoreny:= FALSE;
			P2_Robot.KOM_OUT.GriperMvCase_DrziMVcase:= FALSE;
			P2_Robot.KOM_OUT.GriperMvCase_DrziPowerCP:= FALSE;
			P2_Robot.KOM_OUT.GriperMvCase_Zatvoreny:= TRUE;
		ELSE
			P2_Robot.KOM_OUT.GriperMvCase_Otvoreny:= FALSE;
			P2_Robot.KOM_OUT.GriperMvCase_DrziMVcase:= FALSE;
			P2_Robot.KOM_OUT.GriperMvCase_DrziPowerCP:= FALSE;
			P2_Robot.KOM_OUT.GriperMvCase_Zatvoreny:= FALSE;
		END_IF
	ELSIF P2_Robot.KOM_OUT.TypGripra_5H THEN
		IF P2_Robot.PAR.Griper_4F_5F_5H_IOLink_Inputs <= 30 THEN
			P2_Robot.KOM_OUT.Griper5H_Zatvoreny:= FALSE;
			P2_Robot.KOM_OUT.Griper5H_DrziBusbary:= FALSE;
			P2_Robot.KOM_OUT.Griper5H_Otvoreny:= TRUE;
		ELSIF P2_Robot.PAR.Griper_4F_5F_5H_IOLink_Inputs >= 880 AND P2_Robot.PAR.Griper_4F_5F_5H_IOLink_Inputs <= 897 THEN
			P2_Robot.KOM_OUT.Griper5H_Zatvoreny:= FALSE;
			P2_Robot.KOM_OUT.Griper5H_Otvoreny:= FALSE;
			P2_Robot.KOM_OUT.Griper5H_DrziBusbary:= TRUE;
		ELSIF P2_Robot.PAR.Griper_4F_5F_5H_IOLink_Inputs >= 992 THEN
			P2_Robot.KOM_OUT.Griper5H_Otvoreny:= FALSE;
			P2_Robot.KOM_OUT.Griper5H_DrziBusbary:= FALSE;
			P2_Robot.KOM_OUT.Griper5H_Zatvoreny:= TRUE;
		ELSE
			P2_Robot.KOM_OUT.Griper5H_Otvoreny:= FALSE;
			P2_Robot.KOM_OUT.Griper5H_DrziBusbary:= FALSE;
			P2_Robot.KOM_OUT.Griper5H_Zatvoreny:= FALSE;
		END_IF
	ELSE
		P2_Robot.KOM_OUT.Griper4F_Otvoreny:= FALSE;
		P2_Robot.KOM_OUT.Griper4F_DrziBusbary:= FALSE;
		P2_Robot.KOM_OUT.Griper4F_Zatvoreny:= FALSE;
		P2_Robot.KOM_OUT.GriperMvCase_Otvoreny:= FALSE;
		P2_Robot.KOM_OUT.GriperMvCase_DrziMVcase:= FALSE;
		P2_Robot.KOM_OUT.GriperMvCase_DrziPowerCP:= FALSE;
		P2_Robot.KOM_OUT.GriperMvCase_Zatvoreny:= FALSE;
		P2_Robot.KOM_OUT.Griper5H_Otvoreny:= FALSE;
		P2_Robot.KOM_OUT.Griper5H_DrziBusbary:= FALSE;
		P2_Robot.KOM_OUT.Griper5H_Zatvoreny:= FALSE;
	END_IF

		END_ACTION
```

#### ProfinetKomunikaciaRobot.st
```iecst
ACTION ProfinetKomunikaciaRobot:

	//Vstupy z Robota do PLC//
	P2_Robot.KOM_IN.Stav_RezimAUTOMAT:= P2_Robot.KOM_IN.Profinet_PLC_INPUTS[0].0;
	P2_Robot.KOM_IN.Stav_ProgramRUN:= P2_Robot.KOM_IN.Profinet_PLC_INPUTS[0].1;
	P2_Robot.KOM_IN.Stav_MotoryOFF:= P2_Robot.KOM_IN.Profinet_PLC_INPUTS[0].2;
	P2_Robot.KOM_IN.Stav_MotoryON:= P2_Robot.KOM_IN.Profinet_PLC_INPUTS[0].3;
	P2_Robot.KOM_IN.Stav_RobotCS:= P2_Robot.KOM_IN.Profinet_PLC_INPUTS[0].4;
	P2_Robot.KOM_IN.Profinet_PLC_INPUTS[0].5;
	P2_Robot.KOM_IN.Profinet_PLC_INPUTS[0].6;
	P2_Robot.KOM_IN.Profinet_PLC_INPUTS[0].7;

	P2_Robot.OUT.ZatvorGriper_YV4:= P2_Robot.KOM_IN.Profinet_PLC_INPUTS[1].0;
	P2_Robot.OUT.OtvorGriper_YV3:= P2_Robot.KOM_IN.Profinet_PLC_INPUTS[1].1;
	P2_Robot.OUT.ZaistiGriper_YV1:= P2_Robot.KOM_IN.Profinet_PLC_INPUTS[1].2;
	P2_Robot.OUT.OdistiGriper_YV2:= P2_Robot.KOM_IN.Profinet_PLC_INPUTS[1].3;
	P2_Robot.OUT.ZapniVakum5H_YV8:= P2_Robot.KOM_IN.Profinet_PLC_INPUTS[1].4;
	P2_Robot.OUT.ZapniVakum4F5F_YV6:= P2_Robot.KOM_IN.Profinet_PLC_INPUTS[1].5;
	P2_Robot.KOM_IN.Stav_Busbary5H_Odobrate:= P2_Robot.KOM_IN.Profinet_PLC_INPUTS[1].6;
	P2_Robot.KOM_IN.Stav_Busbary5F_Odobrate:= P2_Robot.KOM_IN.Profinet_PLC_INPUTS[1].7;

	P2_Robot.KOM_IN.Stav_Busbary4F_Odobrate:= P2_Robot.KOM_IN.Profinet_PLC_INPUTS[2].0;
	P2_Robot.KOM_IN.Stav_Busbary5H_Polozene:= P2_Robot.KOM_IN.Profinet_PLC_INPUTS[2].1;
	P2_Robot.KOM_IN.Stav_Busbary5F_Polozene:= P2_Robot.KOM_IN.Profinet_PLC_INPUTS[2].2;
	P2_Robot.KOM_IN.Stav_Busbary4F_Polozene:= P2_Robot.KOM_IN.Profinet_PLC_INPUTS[2].3;
	P2_Robot.KOM_IN.Stav_RobotPoziciaCakania:= P2_Robot.KOM_IN.Profinet_PLC_INPUTS[2].4;
	P2_Robot.KOM_IN.Stav_Filter5H_Dotlaceny:= P2_Robot.KOM_IN.Profinet_PLC_INPUTS[2].5;
	P2_Robot.KOM_IN.Profinet_PLC_INPUTS[2].6;
	P2_Robot.KOM_IN.Stav_Cistenie_PowerCP_Odobrate:= P2_Robot.KOM_IN.Profinet_PLC_INPUTS[2].7;

	P2_Robot.KOM_IN.Profinet_PLC_INPUTS[3].0;
	P2_Robot.KOM_IN.Profinet_PLC_INPUTS[3].1;
	P2_Robot.KOM_IN.Stav_Cistenie_Otacanie_Ukoncene:= P2_Robot.KOM_IN.Profinet_PLC_INPUTS[3].2;
	P2_Robot.KOM_IN.Stav_Cistenie_PowerCP_v_Cisteni:= P2_Robot.KOM_IN.Profinet_PLC_INPUTS[3].3;
	P2_Robot.KOM_IN.Stav_Cistenie_PowerCP_Polozene:= P2_Robot.KOM_IN.Profinet_PLC_INPUTS[3].4;
	P2_Robot.KOM_IN.Profinet_PLC_INPUTS[3].5;
	P2_Robot.KOM_IN.Profinet_PLC_INPUTS[3].6;
	P2_Robot.KOM_IN.Stav_LavyMvCase5H_Odobraty:= P2_Robot.KOM_IN.Profinet_PLC_INPUTS[3].7;

	P2_Robot.KOM_IN.Stav_LavyMvCase5F_Odobraty:= P2_Robot.KOM_IN.Profinet_PLC_INPUTS[4].0;
	P2_Robot.KOM_IN.Stav_LavyMvCase4F_Odobraty:= P2_Robot.KOM_IN.Profinet_PLC_INPUTS[4].1;
	P2_Robot.KOM_IN.Stav_PravyMvCase5H_Odobraty:= P2_Robot.KOM_IN.Profinet_PLC_INPUTS[4].2;
	P2_Robot.KOM_IN.Stav_PravyMvCase5F_Odobraty:= P2_Robot.KOM_IN.Profinet_PLC_INPUTS[4].3;
	P2_Robot.KOM_IN.Stav_PravyMvCase4F_Odobraty:= P2_Robot.KOM_IN.Profinet_PLC_INPUTS[4].4;
	P2_Robot.KOM_IN.Stav_TopCover5H_Odobraty:= P2_Robot.KOM_IN.Profinet_PLC_INPUTS[4].5;
	P2_Robot.KOM_IN.Stav_TopCover5F_Odobraty:= P2_Robot.KOM_IN.Profinet_PLC_INPUTS[4].6;
	P2_Robot.KOM_IN.Stav_TopCover4F_Odobraty:= P2_Robot.KOM_IN.Profinet_PLC_INPUTS[4].7;

	P2_Robot.OUT.VypniVakum5H_YV9:= P2_Robot.KOM_IN.Profinet_PLC_INPUTS[5].0;
	P2_Robot.OUT.VypniVakum4F5F_YV7:= P2_Robot.KOM_IN.Profinet_PLC_INPUTS[5].1;
	P2_Robot.OUT.OdvzdusnenieVyvodov_YV70:= P2_Robot.KOM_IN.Profinet_PLC_INPUTS[5].2;
	P2_Robot.KOM_IN.Stav_LavyMvCase5H_Polozeny:= P2_Robot.KOM_IN.Profinet_PLC_INPUTS[5].3;
	P2_Robot.KOM_IN.Stav_LavyMvCase5F_Polozeny:= P2_Robot.KOM_IN.Profinet_PLC_INPUTS[5].4;
	P2_Robot.KOM_IN.Stav_LavyMvCase4F_Polozeny:= P2_Robot.KOM_IN.Profinet_PLC_INPUTS[5].5;
	P2_Robot.KOM_IN.Stav_PravyMvCase5H_Polozeny:= P2_Robot.KOM_IN.Profinet_PLC_INPUTS[5].6;
	P2_Robot.KOM_IN.Stav_PravyMvCase5F_Polozeny:= P2_Robot.KOM_IN.Profinet_PLC_INPUTS[5].7;

	P2_Robot.KOM_IN.Stav_PravyMvCase4F_Polozeny:= P2_Robot.KOM_IN.Profinet_PLC_INPUTS[6].0;
	P2_Robot.KOM_IN.Stav_TopCover5H_Polozeny:= P2_Robot.KOM_IN.Profinet_PLC_INPUTS[6].1;
	P2_Robot.KOM_IN.Stav_TopCover5F_Polozeny:= P2_Robot.KOM_IN.Profinet_PLC_INPUTS[6].2;
	P2_Robot.KOM_IN.Stav_TopCover4F_Polozeny:= P2_Robot.KOM_IN.Profinet_PLC_INPUTS[6].3;
	P2_Robot.KOM_IN.Stav_RobotOdparkovany:= P2_Robot.KOM_IN.Profinet_PLC_INPUTS[6].4;
	P2_Robot.KOM_IN.Stav_RobotBezpPozicia_Srobovanie:= P2_Robot.KOM_IN.Profinet_PLC_INPUTS[6].5;
	P2_Robot.KOM_IN.Stav_RobotBezpPozicia_Zvaranie:= P2_Robot.KOM_IN.Profinet_PLC_INPUTS[6].6;
	P2_Robot.KOM_IN.Stav_VystupyZresetovane:= P2_Robot.KOM_IN.Profinet_PLC_INPUTS[6].7;

	P2_Robot.KOM_IN.Stav_BusbaryUvolnene:= P2_Robot.KOM_IN.Profinet_PLC_INPUTS[7].0;
    P2_Robot.KOM_IN.Stav_Griper4F5F_Vymeneny:= P2_Robot.KOM_IN.Profinet_PLC_INPUTS[7].1;
    P2_Robot.KOM_IN.Stav_Griper5H_Vymeneny:= P2_Robot.KOM_IN.Profinet_PLC_INPUTS[7].2;
    P2_Robot.KOM_IN.Stav_GriperCistenia_Vymeneny:= P2_Robot.KOM_IN.Profinet_PLC_INPUTS[7].3;
	P2_Robot.KOM_IN.Stav_RobotOdoberaCover:= P2_Robot.KOM_IN.Profinet_PLC_INPUTS[7].4;

	//Vystupy z PLC do Robota//
	P2_Robot.KOM_OUT.Profinet_PLC_OUTPUTS[0].0:= P2_Robot.KOM_OUT.VypniMotory;
	P2_Robot.KOM_OUT.Profinet_PLC_OUTPUTS[0].1:= P2_Robot.KOM_OUT.ZapniMotory;
	P2_Robot.KOM_OUT.Profinet_PLC_OUTPUTS[0].2:= P2_Robot.KOM_OUT.PP_na_Main;
	P2_Robot.KOM_OUT.Profinet_PLC_OUTPUTS[0].3:= P2_Robot.KOM_OUT.StartProgramu;
	P2_Robot.KOM_OUT.Profinet_PLC_OUTPUTS[0].4:= P2_Robot.KOM_OUT.StartProgramuMain;
	P2_Robot.KOM_OUT.Profinet_PLC_OUTPUTS[0].5:= P2_Robot.KOM_OUT.StopProgramu;
	P2_Robot.KOM_OUT.Profinet_PLC_OUTPUTS[0].6:= P2_Robot.KOM_OUT.Reset_CS;
	P2_Robot.KOM_OUT.Profinet_PLC_OUTPUTS[0].7;

	P2_Robot.KOM_OUT.Profinet_PLC_OUTPUTS[1].0:= P2_Robot.KOM_OUT.TypGripra_5H;
	P2_Robot.KOM_OUT.Profinet_PLC_OUTPUTS[1].1:= P2_Robot.KOM_OUT.TypGripra_45F;
	P2_Robot.KOM_OUT.Profinet_PLC_OUTPUTS[1].2:= P2_Robot.KOM_OUT.TypGripra_MV;
	P2_Robot.KOM_OUT.Profinet_PLC_OUTPUTS[1].3:= P2_Robot.KOM_OUT.Griper4F_Otvoreny;
	P2_Robot.KOM_OUT.Profinet_PLC_OUTPUTS[1].4:= P2_Robot.KOM_OUT.Griper4F_DrziBusbary;
	P2_Robot.KOM_OUT.Profinet_PLC_OUTPUTS[1].5:= P2_Robot.KOM_OUT.Griper4F_Zatvoreny;
	P2_Robot.KOM_OUT.Profinet_PLC_OUTPUTS[1].6:= P2_Robot.KOM_OUT.Griper5H_Otvoreny;
	P2_Robot.KOM_OUT.Profinet_PLC_OUTPUTS[1].7:= P2_Robot.KOM_OUT.Griper5H_DrziBusbary;

	P2_Robot.KOM_OUT.Profinet_PLC_OUTPUTS[2].0:= P2_Robot.KOM_OUT.Griper5H_Zatvoreny;
	P2_Robot.KOM_OUT.Profinet_PLC_OUTPUTS[2].1:= P2_Robot.KOM_OUT.GriperMvCase_Otvoreny;
	P2_Robot.KOM_OUT.Profinet_PLC_OUTPUTS[2].2:= P2_Robot.KOM_OUT.GriperMvCase_DrziMVcase;
	P2_Robot.KOM_OUT.Profinet_PLC_OUTPUTS[2].3:= P2_Robot.KOM_OUT.GriperMvCase_DrziPowerCP;
	P2_Robot.KOM_OUT.Profinet_PLC_OUTPUTS[2].4:= P2_Robot.KOM_OUT.GriperMvCase_Zatvoreny;
	P2_Robot.KOM_OUT.Profinet_PLC_OUTPUTS[2].5:= P2_Robot.IN.SnimacVakua_5H_S2;
	P2_Robot.KOM_OUT.Profinet_PLC_OUTPUTS[2].6:= P2_Robot.IN.SnimacVakua_45F_S1;
	P2_Robot.KOM_OUT.Profinet_PLC_OUTPUTS[2].7:= P2_Robot.KOM_OUT.Odober_Busbary5H;

	P2_Robot.KOM_OUT.Profinet_PLC_OUTPUTS[3].0:= P2_Robot.KOM_OUT.Odober_Busbary5F;
	P2_Robot.KOM_OUT.Profinet_PLC_OUTPUTS[3].1:= P2_Robot.KOM_OUT.Odober_Busbary4F;
	P2_Robot.KOM_OUT.Profinet_PLC_OUTPUTS[3].2:= P2_Robot.KOM_OUT.Poloz_Busbary5H;
	P2_Robot.KOM_OUT.Profinet_PLC_OUTPUTS[3].3:= P2_Robot.KOM_OUT.Poloz_Busbary5F;
	P2_Robot.KOM_OUT.Profinet_PLC_OUTPUTS[3].4:= P2_Robot.KOM_OUT.Poloz_Busbary4F;
	P2_Robot.KOM_OUT.Profinet_PLC_OUTPUTS[3].5:= P2_Robot.KOM_OUT.Presun_CakaciaPozicia;
	P2_Robot.KOM_OUT.Profinet_PLC_OUTPUTS[3].6:= P2_Robot.KOM_OUT.Dotlac_Filter5H;
	P2_Robot.KOM_OUT.Profinet_PLC_OUTPUTS[3].7;

	P2_Robot.KOM_OUT.Profinet_PLC_OUTPUTS[4].0:= P2_Robot.KOM_OUT.Cistenie_OdoberPowerCP_5H;
	P2_Robot.KOM_OUT.Profinet_PLC_OUTPUTS[4].1:= P2_Robot.KOM_OUT.Cistenie_OdoberPowerCP_5F;
	P2_Robot.KOM_OUT.Profinet_PLC_OUTPUTS[4].2:= P2_Robot.KOM_OUT.Cistenie_OdoberPowerCP_4F;
	P2_Robot.KOM_OUT.Profinet_PLC_OUTPUTS[4].3;
	P2_Robot.KOM_OUT.Profinet_PLC_OUTPUTS[4].4;
	P2_Robot.KOM_OUT.Profinet_PLC_OUTPUTS[4].5;
	P2_Robot.KOM_OUT.Profinet_PLC_OUTPUTS[4].6:= P2_Robot.KOM_OUT.Cistenie_PolozPowerCP_5H;
	P2_Robot.KOM_OUT.Profinet_PLC_OUTPUTS[4].7:= P2_Robot.KOM_OUT.Cistenie_PolozPowerCP_5F;

	P2_Robot.KOM_OUT.Profinet_PLC_OUTPUTS[5].0:= P2_Robot.KOM_OUT.Cistenie_PolozPowerCP_4F;
	P2_Robot.KOM_OUT.Profinet_PLC_OUTPUTS[5].1:= P2_Robot.KOM_OUT.Odober_LavyMvCase5H;
	P2_Robot.KOM_OUT.Profinet_PLC_OUTPUTS[5].2:= P2_Robot.KOM_OUT.Odober_LavyMvCase5F;
	P2_Robot.KOM_OUT.Profinet_PLC_OUTPUTS[5].3:= P2_Robot.KOM_OUT.Odober_LavyMvCase4F;
	P2_Robot.KOM_OUT.Profinet_PLC_OUTPUTS[5].4:= P2_Robot.KOM_OUT.Odober_PravyMvCase5H;
	P2_Robot.KOM_OUT.Profinet_PLC_OUTPUTS[5].5:= P2_Robot.KOM_OUT.Odober_PravyMvCase5F;
	P2_Robot.KOM_OUT.Profinet_PLC_OUTPUTS[5].6:= P2_Robot.KOM_OUT.Odober_PravyMvCase4F;
	P2_Robot.KOM_OUT.Profinet_PLC_OUTPUTS[5].7:= P2_Robot.KOM_OUT.Odober_TopCover5H;

	P2_Robot.KOM_OUT.Profinet_PLC_OUTPUTS[6].0:= P2_Robot.KOM_OUT.Odober_TopCover5F;
	P2_Robot.KOM_OUT.Profinet_PLC_OUTPUTS[6].1:= P2_Robot.KOM_OUT.Odober_TopCover4F;
	P2_Robot.KOM_OUT.Profinet_PLC_OUTPUTS[6].2:= P2_Robot.IN.DokStanPritGripra_BusBary5H_IS3;
	P2_Robot.KOM_OUT.Profinet_PLC_OUTPUTS[6].3:= P2_Robot.IN.DokStanPritGripra_BusBary45F_IS2;
	P2_Robot.KOM_OUT.Profinet_PLC_OUTPUTS[6].4:= P2_Robot.IN.DokStanPritGripra_MVcase_IS1;
	P2_Robot.KOM_OUT.Profinet_PLC_OUTPUTS[6].5:= P2_Robot.KOM_OUT.Cistenie_BezpecnaPozicia;
	P2_Robot.KOM_OUT.Profinet_PLC_OUTPUTS[6].6:= P2_Robot.KOM_OUT.Cistenie_OtacajPowerCP;
	P2_Robot.KOM_OUT.Profinet_PLC_OUTPUTS[6].7:= P2_Robot.KOM_OUT.ManipSrobovania_BezpecnaPozicia;

	P2_Robot.KOM_OUT.Profinet_PLC_OUTPUTS[7].0:= P2_Robot.KOM_OUT.Poloz_LavyMvCase5H;
	P2_Robot.KOM_OUT.Profinet_PLC_OUTPUTS[7].1:= P2_Robot.KOM_OUT.Poloz_LavyMvCase5F;
	P2_Robot.KOM_OUT.Profinet_PLC_OUTPUTS[7].2:= P2_Robot.KOM_OUT.Poloz_LavyMvCase4F;
	P2_Robot.KOM_OUT.Profinet_PLC_OUTPUTS[7].3:= P2_Robot.KOM_OUT.Poloz_PravyMvCase5H;
	P2_Robot.KOM_OUT.Profinet_PLC_OUTPUTS[7].4:= P2_Robot.KOM_OUT.Poloz_PravyMvCase5F;
	P2_Robot.KOM_OUT.Profinet_PLC_OUTPUTS[7].5:= P2_Robot.KOM_OUT.Poloz_PravyMvCase4F;
	P2_Robot.KOM_OUT.Profinet_PLC_OUTPUTS[7].6:= P2_Robot.KOM_OUT.Poloz_TopCover5H;
	P2_Robot.KOM_OUT.Profinet_PLC_OUTPUTS[7].7:= P2_Robot.KOM_OUT.Poloz_TopCover5F;

	P2_Robot.KOM_OUT.Profinet_PLC_OUTPUTS[8].0:= P2_Robot.KOM_OUT.Poloz_TopCover4F;
	P2_Robot.KOM_OUT.Profinet_PLC_OUTPUTS[8].1:= P2_Robot.KOM_OUT.Odparkovanie;
	P2_Robot.KOM_OUT.Profinet_PLC_OUTPUTS[8].2:= P2_Robot.KOM_OUT.Zvaranie_BezpecnaPozicia;
	P2_Robot.KOM_OUT.Profinet_PLC_OUTPUTS[8].3:= P2_Robot.KOM_OUT.UvolniBusbary;
    P2_Robot.KOM_OUT.Profinet_PLC_OUTPUTS[8].4:= P2_Robot.KOM_OUT.ZmenaGripra_4F5F;
    P2_Robot.KOM_OUT.Profinet_PLC_OUTPUTS[8].5:= P2_Robot.KOM_OUT.ZmenaGripra_5H;
    P2_Robot.KOM_OUT.Profinet_PLC_OUTPUTS[8].6:= P2_Robot.KOM_OUT.ZmenaGripra_Cistenie;
    P2_Robot.KOM_OUT.Profinet_PLC_OUTPUTS[8].7:= P2_Robot.KOM_OUT.ZopakujOdoberanie;

END_ACTION
```

### Program Logical/Program/Pracovisko_2/P2_StoperZvarania (IEC)
